FUNCTION_BLOCK TerminalGroupReport_FB
VAR_INPUT
	Enable 				: BOOL;
	pGroupCtrl			: POINTER TO Terminal_Group_Ctrl_typ ;
	Ref_ev_Module_Event : REFERENCE TO ev_MOTOR_POSITION_ERROR REF= ev_MOTOR_POSITION_ERROR;
END_VAR
VAR_IN_OUT
	In 		: ARRAY[*]OF Terminal_Ctrl_typ ;	
	//Out		: ARRAY[*]OF ErrCollector_Out ;
END_VAR

VAR
	LogMsgInit          : BOOL := TRUE;
	LogMsg_0 			: LogMsg ;
	//Get old events from Q
	ExecuteTrig: 		Trigger;	
	WrongState :   		BOOL;
	nI         : DINT;
	InFault    : BOOL;
	
	fbPrgmBasic :FB_PrgmBasic;
	
	
	//Debug
	intErrorCounter : USINT := 0;
	
	LowerBound         : DINT;
END_VAR






IF pGroupCtrl <> 0 THEN
		
	IF LogMsgInit THEN      
		LogMsgInit := FALSE ;
		fnLogMsgInit(ADR(LogMsg_0), pGroupCtrl^.In.Par.GroupName, ADR(LogGlobalArray), ADR(CONST_ZERO));
		LogMsg_0.Enable:= 		TRUE;
	END_IF

	IF Enable THEN
		InFault := FALSE;
		
		LowerBound := LOWER_BOUND(In,1);
		
		FOR nI:= LOWER_BOUND(In,1) TO UPPER_BOUND(In,1) DO

	
			IF 	In[nI].In.Par.Name <> 'Empty' THEN
							
				// IF already in error reset others status
				IF InFault THEN
					In[nI].Out.Status.Fault := FALSE;
				ELSE	
					//If terminal is not on OPER state
					IF ((In[nI].Out.Status.TerminalState AND eTerminalStates.OP) = 0) THEN
							
						IF In[nI].Out.Status.Active THEN
							InFault := TRUE;												
							
							IF In[nI].Out.Status.Fault = FALSE THEN
								Meth_SetError(nI);							
							END_IF
						ELSE // Module Not Active
							
							Meth_HandleModuleNotActive(nI);										
						END_IF
						In[nI].Out.Status.Fault := TRUE;
					ELSE
						In[nI].Out.Status.Fault := FALSE;		
					END_IF
				
						
				END_IF
				In[nI].Out.Status.Active := 0;
				In[nI].Out.Monitor.SubSysName := '';
			END_IF
			
		END_FOR
		
		IF NOT InFault THEN
			pGroupCtrl^.Out.Status.errorBit := 0;
		END_IF	
		
		// Reset if for was brake	
		In[nI].Out.Status.Active := 0;
		In[nI].Out.Monitor.SubSysName := '';
	END_IF
	
	

END_IF	
fbPrgmBasic();
//fnLogTransfer FUNCTION call
fnLogTransfer(ADR(LogMsg_0));

METHOD Meth_HandleModuleNotActive : BOOL
VAR_INPUT
	
	NonActiveIndex: DINT;
	
END_VAR
VAR
	internalIndex : DINT;
END_VAR
	//if last
	IF NonActiveIndex = UPPER_BOUND(In,1) THEN
		//	System is OK because it is last
					
		//If next is not OK
	ELSIF In[nI+1].Out.Status.TerminalState <> eTerminalStates.OP THEN
		IF In[nI+1].Out.Status.Active THEN
			InFault := TRUE;	
			//next is Active and not OK
			IF In[NonActiveIndex].Out.Status.Fault = FALSE THEN
				Meth_SetError(NonActiveIndex);											
			END_IF											
			InFault := TRUE;
		ELSE// Check if there is active module after the problematic module
			FOR internalIndex:= NonActiveIndex TO UPPER_BOUND(In,1) DO
				IF In[internalIndex].Out.Status.Active THEN
					InFault := TRUE;	
					IF In[NonActiveIndex].Out.Status.Fault = FALSE THEN
						Meth_SetError(NonActiveIndex);											
					END_IF	
				END_IF		
			END_FOR
		END_IF
		
									
	ELSE 
			//Continue the next module is OK	;
		 	
	END_IF
END_METHOD

METHOD Meth_SendEvent : BOOL
VAR_INPUT
	RefEvent : REFERENCE TO EventHelper;
END_VAR
VAR
	EventParameters:EventParam_Typ;	
	EventHeader:EventHeader_Typ;	
	Dummy :DINT :=0;
//	pFlowID :POINTER TO DINT;
END_VAR
IF __ISVALIDREF(RefEvent) THEN
		
		EventHeader.SubsysID :=		pGroupCtrl^.In.Par.GroupID  ; 
 
		EventParameters.MotorID := 		 In[nI].In.Par.ModuleID; 	// Motor ID

		fbPrgmBasic.mEventThrow(RefEvent,ADR(EventHeader),ADR(EventParameters) );			//RefEvent();
		Meth_SendEvent := TRUE;
		
		


		//Debug
		intErrorCounter := intErrorCounter + 1;
		
END_IF
END_METHOD

METHOD Meth_SetError : BOOL
VAR_INPUT
	
	TerminalIndex: DINT;
	
END_VAR
VAR
	BitBase : ULINT ;
END_VAR
Meth_SendEvent(Ref_ev_Module_Event);

fnLogMsg(ADR(LogMsg_0), LOG_INFO, 'Terminal Error Q Send Group ID %d,In[nI].In.Par.ModuleID =%d',
							pGroupCtrl^.In.Par.GroupID  ,
							In[TerminalIndex].In.Par.ModuleID,							
							0);

							
BitBase := 2;			
pGroupCtrl^.Out.Status.errorBit := SHL(BitBase,(TerminalIndex -LowerBound));
END_METHOD

END_FUNCTION_BLOCK

(* stored: Version 1.1.0.1, ProductVersion 3.1.4024.3
   POU TerminalGroupReport_FB: Id {2861ada8-63e0-0302-0267-c182570bf514}, SpecialFunc None
   Method Meth_HandleModuleNotActive: Id {5a9f709d-92a7-033e-393a-2f9bbd539b56}
   Method Meth_SendEvent: Id {eb4303c8-da40-0228-3b13-c421b9fea17c}
   Method Meth_SetError: Id {f59bccd8-d4b7-0dfa-35f2-b4236de5517f} *)
